FUNCTION_BLOCK FB_HMI_TP_BRANCH_B EXTENDS FB_HMI_COMPONENT
VAR_INPUT
END_VAR
VAR_OUTPUT
END_VAR
VAR
END_VAR

END_FUNCTION_BLOCK

(* stored: Version 1.1.0.1, ProductVersion 3.1.4024.14
   POU FB_HMI_TP_BRANCH_B: Id {351926ee-3267-4686-9203-3d7175008f9d}, SpecialFunc None *)
